Fanuc KAREL source: kd00016.KL

-- PROVISIONAL review KL for V770-1; original PC SHA256 80e1582fde0c7b7a67880e73514c804f5f1c9d6b2cf7e8cb41fbbbe6bae7f81f
-- Incomplete behavior may be omitted. Consult companion uncertainty JSON. Do not deploy.
PROGRAM KD00016
%NOLOCKGROUP
VAR
  I : INTEGER
  J : INTEGER
  B : BOOLEAN
  R : REAL
  S : STRING[80]
BEGIN
  -- UNRESOLVED_PC offsets 5-12; opcodes 9C,23
  -- UNRESOLVED_PC offsets 17-24; opcodes 22,62
  -- UNRESOLVED_PC offsets 29-33; opcodes 7F
END KD00016
